{attribute 'GeneratedUsingTerminal: EPP1322-0001-0017'}
{attribute addProperty BoxType "EPP1322-0001-0017"}
{attribute addProperty Id "RC30_AB1_EPP1008_0001EPP1008_78E8D3DD12RC30_AB2_EPP1008_0001EPP1008_78E8D3DD12RC30_AB6_EPP1008_0001EPP1008_78E8D3DD12RC30_AB3_EPP1008_0001EPP1008_78E8D3DD12RC30_AB4_EPP1008_0001EPP1008_78E8D3DD12RC30_AB7_EPP1008_0001EPP1008_78E8D3DD12RC30_AB9_EPP1008_0001EPP1008_78E8D3DD12RC30_AB10_EPP1008_0001EPP1008_78E8D3DD12RC30_AB8_EPP1008_0001EPP1008_78E8D3DD12RC30_AB5_EPP1008_0001EPP1008_78E8D3DD12"}
{attribute addProperty CRC "3990710401"}
{attribute addProperty Size "120"}
{attribute addProperty Name "RC30_EPP (EPP1322-0001)"}
TYPE RC30_EPP_EPP1322_0001_EDDD6881 EXTENDS EPP1322_1FC0878B : STRUCT
    {attribute addProperty Name "RC30_AB1 (EPP1008-0001)"}
    {attribute addProperty PreviousPort "RC30_EPP (EPP1322-0001) : D"}
    {attribute addProperty SyncUnit "C30"}
    RC30_AB1_EPP1008_0001 : EPP1008_78E8D3DD;
    {attribute addProperty Name "RC30_AB2 (EPP1008-0001)"}
    {attribute addProperty PreviousPort "RC30_AB1 (EPP1008-0001) : B"}
    {attribute addProperty SyncUnit "C30"}
    RC30_AB2_EPP1008_0001 : EPP1008_78E8D3DD;
    {attribute addProperty Name "RC30_AB6 (EPP1008-0001)"}
    {attribute addProperty PreviousPort "RC30_AB2 (EPP1008-0001) : B"}
    {attribute addProperty SyncUnit "C30"}
    RC30_AB6_EPP1008_0001 : EPP1008_78E8D3DD;
    {attribute addProperty Name "RC30_AB3 (EPP1008-0001)"}
    {attribute addProperty PreviousPort "RC30_AB6 (EPP1008-0001) : B"}
    {attribute addProperty SyncUnit "C30"}
    RC30_AB3_EPP1008_0001 : EPP1008_78E8D3DD;
    {attribute addProperty Name "RC30_AB4 (EPP1008-0001)"}
    {attribute addProperty PreviousPort "RC30_AB3 (EPP1008-0001) : B"}
    {attribute addProperty SyncUnit "C30"}
    RC30_AB4_EPP1008_0001 : EPP1008_78E8D3DD;
    {attribute addProperty Name "RC30_AB7 (EPP1008-0001)"}
    {attribute addProperty PreviousPort "RC30_EPP (EPP1322-0001) : B"}
    {attribute addProperty SyncUnit "C30"}
    RC30_AB7_EPP1008_0001 : EPP1008_78E8D3DD;
    {attribute addProperty Name "RC30_AB9 (EPP1008-0001)"}
    {attribute addProperty PreviousPort "RC30_AB7 (EPP1008-0001) : B"}
    {attribute addProperty SyncUnit "C30"}
    RC30_AB9_EPP1008_0001 : EPP1008_78E8D3DD;
    {attribute addProperty Name "RC30_AB10 (EPP1008-0001)"}
    {attribute addProperty PreviousPort "RC30_AB9 (EPP1008-0001) : B"}
    {attribute addProperty SyncUnit "C30"}
    RC30_AB10_EPP1008_0001 : EPP1008_78E8D3DD;
    {attribute addProperty Name "RC30_AB8 (EPP1008-0001)"}
    {attribute addProperty PreviousPort "RC30_AB10 (EPP1008-0001) : B"}
    {attribute addProperty SyncUnit "C30"}
    RC30_AB8_EPP1008_0001 : EPP1008_78E8D3DD;
    {attribute addProperty Name "RC30_AB5 (EPP1008-0001)"}
    {attribute addProperty PreviousPort "RC30_AB8 (EPP1008-0001) : B"}
    {attribute addProperty SyncUnit "C30"}
    RC30_AB5_EPP1008_0001 : EPP1008_78E8D3DD;
END_STRUCT
END_TYPE

(* stored: Version 1.2.0.0, ProductVersion 3.1.4024.11
   DUT RC30_EPP_EPP1322_0001_EDDD6881: Id {9786602c-17d4-0824-08d6-f0e50c13b995} *)
